Omron CX-Programmer project NewProject (CX-Programmer 9.75)

# PLC MIXER_PROJECT: CJ2M CPU11

## Global symbols (name address type ; comment)
0.00 BOOL  ; START
0.01 BOOL  ; LLS
0.02 BOOL  ; MLS
0.03 BOOL  ; HLS
0.04 BOOL  ; TEMP SENSOR
100.00 BOOL  ; IV1
100.01 BOOL  ; IV2
100.02 BOOL  ; MIXER
100.03 BOOL  ; BOILER
100.04 BOOL  ; OUTLET
T0000 BOOL  ; T0

## Program NewProgram1 (cyclic task 0)

### Section Section1

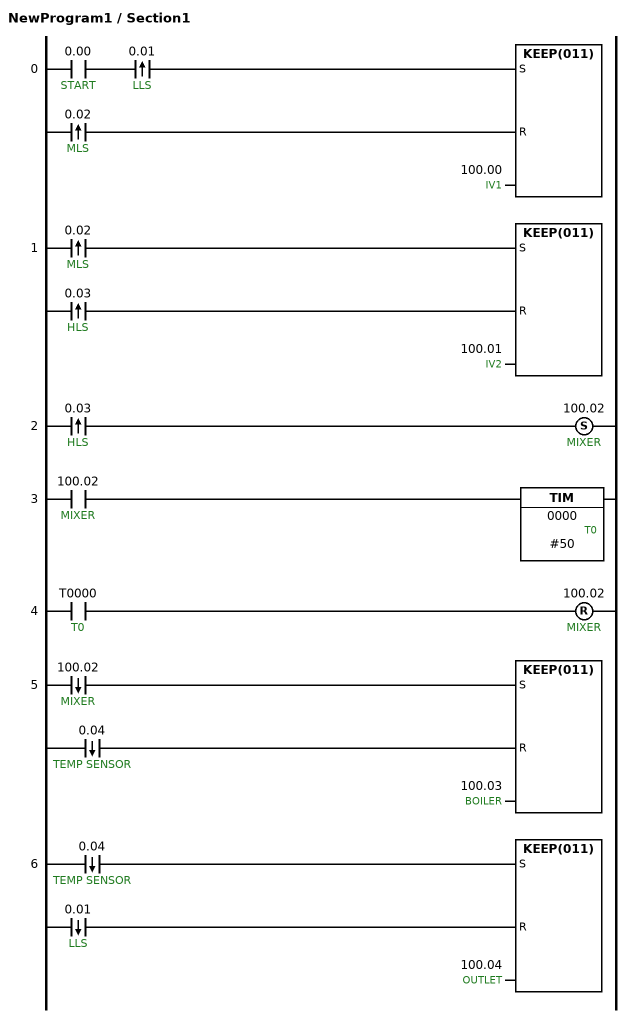
; rung 0
LD 0.00  ; START
@AND 0.01  ; LLS
@LD 0.02  ; MLS
KEEP(011) 100.00  ; IV1
; rung 1
@LD 0.02  ; MLS
@LD 0.03  ; HLS
KEEP(011) 100.01  ; IV2
; rung 2
@LD 0.03  ; HLS
SET 100.02  ; MIXER
; rung 3
LD 100.02  ; MIXER
TIM 0000 #50  ; T0
; rung 4
LD T0000  ; T0
RSET 100.02  ; MIXER
; rung 5
%LD 100.02  ; MIXER
%LD 0.04  ; TEMP SENSOR
KEEP(011) 100.03  ; BOILER
; rung 6
%LD 0.04  ; TEMP SENSOR
%LD 0.01  ; LLS
KEEP(011) 100.04  ; OUTLET

### Section END
; rung 0
END(001)